// TwinCAT 3 PLC project ProbeZPlc
// ProgramVersion: 3.1.4024.12
// libraries:
//   Tc2_MC2, * (Beckhoff Automation GmbH)
//   Tc2_Standard, * (Beckhoff Automation GmbH)
//   Tc2_System, * (Beckhoff Automation GmbH)
//   Tc3_Module, * (Beckhoff Automation GmbH)
// project tree:
//   DUTs/ XY_Stage_State.TcDUT
//   / PlcTask.TcTTO
//   POUs/ MAIN.TcPOU
// real-time tasks:
//   TASK PlcTask: cycle T#10ms, priority 20, ADS port 350
// motion (NC):
//   TASK NC-Task 1 SAF: cycle T#2ms, priority 4, ADS port 501
//   TASK NC-Task 1 SVB: cycle T#10ms, priority 8, ADS port 511
//   AXIS Axis 1 (id 1)
//     OtherSettings: AllowMotionCmdToSlave=true
//     encoder EncType=19
//       EncPara: MaxCount=#xffffffff
//     drive DrvType=16
//       DrvPara: MaxCount=#xffffffff, DriveControlDWord=#x00020000
//         Analog: TorqueSetpointScale=10, ScaleFactorActTorque=0.1
//         TimeComp: TaskDelayCycles=1
//     controller CtrType=1
//       CtrPara: PriorControlFactor=1
//         Observer: BandWidth=20
//   AXIS Axis 2 (id 2)
//     OtherSettings: AllowMotionCmdToSlave=true
//     encoder EncType=19
//       EncPara: MaxCount=#xffffffff
//     drive DrvType=16
//       DrvPara: MaxCount=#xffffffff, DriveControlDWord=#x00020000
//         Analog: TorqueSetpointScale=10, ScaleFactorActTorque=0.1
//         TimeComp: TaskDelayCycles=1
//     controller CtrType=1
//       CtrPara: PriorControlFactor=1
//         Observer: BandWidth=20
//   AXIS Axis 3 (id 3)
//     General: UnitName=°
//     Dynamic: Acceleration=10116, Deceleration=10116, Jerk=30348
//     Velo: RefSearch=67.44, RefSync=67.44, SlowManual=337.2, FastManual=2023.2, Fast=6744, Maximum=6744
//     OtherSettings: AllowMotionCmdToSlave=true
//     encoder EncType=19
//       EncPara: ScaleFactorNumerator=360, ScaleFactorDenominator=1048576, MaxCount=#xffffffff
//     drive DrvType=16
//       DrvPara: MaxCount=#xffffffff, DriveControlDWord=#x00020100
//         Analog: VeloReferenz=7418.4, VeloScale=32, TorqueSetpointScale=10, ScaleFactorActTorque=0.1
//         TimeComp: TaskDelayCycles=1
//     controller CtrType=1
//       CtrPara: PriorControlFactor=1
//         PosDiffControl: Enable=false
//         Observer: BandWidth=20
//   AXIS Axis 4 (id 4)
//     General: UnitName=°
//     Dynamic: Acceleration=10116, Deceleration=10116, Jerk=30348
//     Velo: RefSearch=67.44, RefSync=67.44, SlowManual=337.2, FastManual=2023.2, Fast=6744, Maximum=6744
//     OtherSettings: AllowMotionCmdToSlave=true
//     encoder EncType=19
//       EncPara: ScaleFactorNumerator=360, ScaleFactorDenominator=1048576, MaxCount=#xffffffff
//     drive DrvType=16
//       DrvPara: MaxCount=#xffffffff, DriveControlDWord=#x00020100
//         Analog: VeloReferenz=7418.4, VeloScale=32, TorqueSetpointScale=10, ScaleFactorActTorque=0.1
//         TimeComp: TaskDelayCycles=1
//     controller CtrType=1
//       CtrPara: PriorControlFactor=1
//         PosDiffControl: Enable=false
//         Observer: BandWidth=20
// I/O:
//   DEVICE Device 1 (EtherCAT), AmsNetId 192.168.1.235.2.1
//     Term 1 (EK1200) [EK1200-5000 EtherCAT Power supply (2A E-Bus)]
//       Term 2 (EK1110) [EK1110 EtherCAT extension]
//     Term 3 (EK1100) [EK1100 EtherCAT Coupler (2A E-Bus)]
//       Term 4 (EL4134) [EL4134 4Ch. Ana. Output -10/+10V, 16bit]
//       Term 5 (EL3104) [EL3104 4Ch. Ana. Input +/-10V Diff.]
//       Term 6 (EL7201-0010) [EL7201-0010 1Ch. MDP742 Servo motor output stage with OCT (50V, 2.8A RMS)]
//       Term 7 (EL5032) [EL5032 2Ch. EnDat Encoder]
//       Term 8 (EL1889) [EL1889 16Ch. Dig. Input 24V, 3ms, negative]
//       Term 9 (EL7201-0010) [EL7201-0010 1Ch. MDP742 Servo motor output stage with OCT (50V, 2.8A RMS)]
//       Term 10 (EL7221-9014) [EL7221-9014 1Ch. MDP742 Servo motor output stage with OCT (50V, 8A RMS) and STO input]
//       Term 11 (EL7221-9014) [EL7221-9014 1Ch. MDP742 Servo motor output stage with OCT (50V, 8A RMS) and STO input]
//       Term 12 (EL2634) [EL2634 4Ch. Relay Output, NO (250V AC / 30V DC)]
//       Term 13 (EL9011) [EL9011 End Terminal]
// variable links:
//   NC-Task 1 SAF/Axes/Axis 1 <-> Device 1 (EtherCAT)/Term 3 (EK1100)/Term 6 (EL7201-0010)
//     Drive/Inputs/In/nDcOutputTime <-> InfoData/DcOutputShift
//     Drive/Inputs/In/nState1 <-> DRV Statusword/Statusword
//     Drive/Inputs/In/nState2 <-> DRV Statusword/Statusword @bit 8
//     Drive/Inputs/In/nState4 @bit 1 <-> WcState/InputToggle
//     Drive/Inputs/In/nState4 <-> WcState/WcState
//     Drive/Outputs/Out/nCtrl1 <-> DRV Controlword/Controlword
//     Drive/Outputs/Out/nCtrl2 <-> DRV Controlword/Controlword @bit 8
//     Drive/Outputs/Out/nDataOut2 <-> DRV Target velocity/Target velocity
//     Enc/Inputs/In/nDataIn1 <-> FB Position/Position
//     Enc/Inputs/In/nDcInputTime <-> InfoData/DcInputShift
//     Enc/Inputs/In/nState4 @bit 1 <-> WcState/InputToggle
//     Enc/Inputs/In/nState4 <-> WcState/WcState
//   NC-Task 1 SAF/Axes/Axis 2 <-> Device 1 (EtherCAT)/Term 3 (EK1100)/Term 9 (EL7201-0010)
//     Drive/Inputs/In/nDcOutputTime <-> InfoData/DcOutputShift
//     Drive/Inputs/In/nState1 <-> DRV Statusword/Statusword
//     Drive/Inputs/In/nState2 <-> DRV Statusword/Statusword @bit 8
//     Drive/Inputs/In/nState4 @bit 1 <-> WcState/InputToggle
//     Drive/Inputs/In/nState4 <-> WcState/WcState
//     Drive/Outputs/Out/nCtrl1 <-> DRV Controlword/Controlword
//     Drive/Outputs/Out/nCtrl2 <-> DRV Controlword/Controlword @bit 8
//     Drive/Outputs/Out/nDataOut2 <-> DRV Target velocity/Target velocity
//     Enc/Inputs/In/nDataIn1 <-> FB Position/Position
//     Enc/Inputs/In/nDcInputTime <-> InfoData/DcInputShift
//     Enc/Inputs/In/nState4 @bit 1 <-> WcState/InputToggle
//     Enc/Inputs/In/nState4 <-> WcState/WcState
//   NC-Task 1 SAF/Axes/Axis 3 <-> Device 1 (EtherCAT)/Term 3 (EK1100)/Term 10 (EL7221-9014)
//     Drive/Inputs/In/nDataIn1 <-> DRV Following error actual value/Following error actual value
//     Drive/Inputs/In/nDcOutputTime <-> InfoData/DcOutputShift
//     Drive/Inputs/In/nState1 <-> DRV Statusword/Statusword
//     Drive/Inputs/In/nState2 <-> DRV Statusword/Statusword @bit 8
//     Drive/Inputs/In/nState4 @bit 1 <-> WcState/InputToggle
//     Drive/Inputs/In/nState4 <-> WcState/WcState
//     Drive/Outputs/Out/nCtrl1 <-> DRV Controlword/Controlword
//     Drive/Outputs/Out/nCtrl2 <-> DRV Controlword/Controlword @bit 8
//     Drive/Outputs/Out/nDataOut1 <-> DRV Target position/Target position
//     Enc/Inputs/In/nDataIn1 <-> FB Position/Position
//     Enc/Inputs/In/nDcInputTime <-> InfoData/DcInputShift
//     Enc/Inputs/In/nState4 @bit 1 <-> WcState/InputToggle
//     Enc/Inputs/In/nState4 <-> WcState/WcState
//   NC-Task 1 SAF/Axes/Axis 4 <-> Device 1 (EtherCAT)/Term 3 (EK1100)/Term 11 (EL7221-9014)
//     Drive/Inputs/In/nDataIn1 <-> DRV Following error actual value/Following error actual value
//     Drive/Inputs/In/nDcOutputTime <-> InfoData/DcOutputShift
//     Drive/Inputs/In/nState1 <-> DRV Statusword/Statusword
//     Drive/Inputs/In/nState2 <-> DRV Statusword/Statusword @bit 8
//     Drive/Inputs/In/nState4 @bit 1 <-> WcState/InputToggle
//     Drive/Inputs/In/nState4 <-> WcState/WcState
//     Drive/Outputs/Out/nCtrl1 <-> DRV Controlword/Controlword
//     Drive/Outputs/Out/nCtrl2 <-> DRV Controlword/Controlword @bit 8
//     Drive/Outputs/Out/nDataOut1 <-> DRV Target position/Target position
//     Enc/Inputs/In/nDataIn1 <-> FB Position/Position
//     Enc/Inputs/In/nDcInputTime <-> InfoData/DcInputShift
//     Enc/Inputs/In/nState4 @bit 1 <-> WcState/InputToggle
//     Enc/Inputs/In/nState4 <-> WcState/WcState
//   ProbeZPlc/ProbeZPlc Instance <-> NC-Task 1 SAF/Axes/Axis 3
//     PlcTask Inputs/MAIN.axisX.NcToPlc <-> Outputs/ToPlc
//     PlcTask Outputs/MAIN.axisX.PlcToNc <-> Inputs/FromPlc
//   ProbeZPlc/ProbeZPlc Instance <-> NC-Task 1 SAF/Axes/Axis 4
//     PlcTask Inputs/MAIN.axisY.NcToPlc <-> Outputs/ToPlc
//     PlcTask Outputs/MAIN.axisY.PlcToNc <-> Inputs/FromPlc

CONFIGURATION ProbeZPlc
    RESOURCE PLC ON TwinCAT3
        TASK PlcTask(INTERVAL := T#10ms, PRIORITY := 20);
        PROGRAM MAIN WITH PlcTask : MAIN;
    END_RESOURCE
END_CONFIGURATION

// ---- DUTs/XY_Stage_State.TcDUT
{attribute 'qualified_only'}
{attribute 'strict'}
TYPE XY_Stage_State :
(
	off := 0,
	reset := 1,
	ready := 2,
	moving := 3,
	error := 9
);
END_TYPE

// ---- POUs/MAIN.TcPOU
PROGRAM MAIN
VAR
	{attribute 'OPC.UA.DA' := '1'}
	state: XY_Stage_State; (* XY Stage State *)
	
	// motor variables
	axisX		: AXIS_REF;
	axisY		: AXIS_REF;
	fbXReset	: MC_Reset;
	fbYReset	: MC_Reset;
	fbXPower	: MC_Power;
	fbYPower	: MC_Power;
	fbXMoveAbs	: MC_MoveAbsolute;
	fbYMoveAbs	: MC_MoveAbsolute;
	bReset		: BOOL := FALSE;
	bXEnable	: BOOL := FALSE;
	bYEnable	: BOOL := FALSE;
	bMove		: BOOL := FALSE;
	fXTargetPos	: LREAL := 0;
	fYTargetPos : LREAL := 0;
	fXTargetVel : LREAL := 360;
	fYTargetVel : LREAL := 360;
	
	// inputs
	{attribute 'OPC.UA.DA' := '1'}
	inputXPos	: LREAL := 0;
	{attribute 'OPC.UA.DA' := '1'}
	inputYPos	: LREAL := 0;
	{attribute 'OPC.UA.DA' := '1'}
	inputXVel	: LREAL := 360;
	{attribute 'OPC.UA.DA' := '1'}
	inputYVel	: LREAL := 360;
	
	// outputs
	{attribute 'OPC.UA.DA' := '1'}
	{attribute 'OPC.UA.DA.Access' := '1'}
	XPos		: LREAL; (* X position *)
	{attribute 'OPC.UA.DA' := '1'}
	{attribute 'OPC.UA.DA.Access' := '1'}
	YPos		: LREAL; (* Y position *)
	{attribute 'OPC.UA.DA' := '1'}
	{attribute 'OPC.UA.DA.Access' := '1'}
	XVel		: LREAL; (* X velocity *)
	{attribute 'OPC.UA.DA' := '1'}
	{attribute 'OPC.UA.DA.Access' := '1'}
	YVel		: LREAL; (* Y velocity *)
	{attribute 'OPC.UA.DA' := '1'}
	{attribute 'OPC.UA.DA.Access' := '1'}
	XLag		: LREAL := 0; (* X position lag *)
	{attribute 'OPC.UA.DA' := '1'}
	{attribute 'OPC.UA.DA.Access' := '1'}
	YLag		: LREAL := 0; (* Y position lag *)
	{attribute 'OPC.UA.DA' := '1'}
	{attribute 'OPC.UA.DA.Access' := '1'}
	XLagMax		: LREAL := 0; (* maximum X position lag (abs val) *)
	{attribute 'OPC.UA.DA' := '1'}
	{attribute 'OPC.UA.DA.Access' := '1'}
	YLagMax		: LREAL := 0; (* maximum Y position lag (abs val) *)
	{attribute 'OPC.UA.DA' := '1'}
	{attribute 'OPC.UA.DA.Access' := '1'}
	XErrorCode		: UDINT := 0; (* last error code for X *)
	{attribute 'OPC.UA.DA' := '1'}
	{attribute 'OPC.UA.DA.Access' := '1'}
	YErrorCode		: UDINT := 0; (* last error code for Y *)
	
END_VAR

axisX.ReadStatus();
axisY.ReadStatus();

// process input & output variables
// these limits taken from Drive Manager
inputXVel := MIN(inputXVel, 6744);
inputYVel := MIN(inputYVel, 6744);

XPos := axisX.NcToPlc.ActPos;
YPos := axisY.NcToPlc.ActPos;
XVel := axisX.NcToPlc.ActVelo;
YVel := axisY.NcToPlc.ActVelo;
XLag := axisX.NcToPlc.PosDiff;
YLag := axisY.NcToPlc.PosDiff;
XLagMax := MAX(ABS(XLag), XLagMax);
YLagMax := MAX(ABS(YLag), YLagMax);

IF axisX.Status.Error = TRUE OR axisY.Status.Error = TRUE OR
	fbXPower.Error = TRUE OR fbYPower.Error = TRUE OR
	fbXMoveAbs.Error = TRUE OR fbYMoveAbs.Error = TRUE THEN
	XErrorCode := MAX(axisX.Status.ErrorID, fbXPower.ErrorID, fbXMoveAbs.ErrorID);
	YErrorCode := MAX(axisY.Status.ErrorID, fbYPower.ErrorID, fbYMoveAbs.ErrorID);
	state := XY_Stage_State.error;
END_IF

CASE state OF
XY_Stage_State.off: // init (power off)
	bReset := FALSE;
	bXEnable := FALSE;
	bYEnable := FALSE;
	bMove := FALSE;
XY_Stage_State.reset: // reset & enable power to axes
	bReset := TRUE;
	bXEnable := FALSE; // FIX temporary
	bYEnable := TRUE;
	XErrorCode := 0;
	YErrorCode := 0;
	IF fbXReset.Done = TRUE AND fbYReset.Done = TRUE AND
		// FIX fbXPower.Status = TRUE AND fbYPower.Status = TRUE THEN
		fbYPower.Status = TRUE THEN
		bReset := FALSE;
		state := XY_Stage_State.ready;
	END_IF
XY_Stage_State.ready: // set up move
	fXTargetPos := inputXPos;
	fYTargetPos := inputYPos;
	fXTargetVel := inputXVel;
	fYTargetVel := inputYVel;
	bMove := TRUE;
	state := XY_Stage_State.moving;
XY_Stage_State.moving: // moving
	// FIX IF fbXMoveAbs.Done = TRUE AND fbYMoveAbs.Done = TRUE THEN
	IF fbYMoveAbs.Done = TRUE THEN
		bMove := FALSE;
		state := XY_Stage_State.ready;
	END_IF
XY_Stage_State.error: // error
	RETURN; // lock into this state
END_CASE

// function blocks, execution controlled by their execute bits
fbXReset(Axis := axisX, Execute := bReset);
fbYReset(Axis := axisY, Execute := bReset);

fbXPower(
	Axis := axisX,
	Enable := bXEnable,
	Enable_Positive := bXEnable,
	Enable_Negative := bXEnable,
	Override := 100);
fbYPower(
	Axis := axisY,
	Enable := bYEnable,
	Enable_Positive := bYEnable,
	Enable_Negative := bYEnable,
	Override := 100);
	
fbXMoveAbs(
	Axis:= axisX,
	Execute:= bMove,
	Position:= fXTargetPos,
	Velocity:= fXTargetVel,
	Acceleration:= ,
	Deceleration:= ,
	Jerk:= );
fbYMoveAbs(
	Axis:= axisY,
	Execute:= bMove,
	Position:= fYTargetPos,
	Velocity:= fYTargetVel,
	Acceleration:= ,
	Deceleration:= ,
	Jerk:= );

END_PROGRAM
